(* IEC 61131-3 sources: osaicnc/ (part 2) *)

(* ---- F_SetRapidOverride.st ---- *)
(*[[
    UserText1= "V15.7",
]]*)
FUNCTION F_SetRapidOverride : DWORD
(*
F ***************************************************************************************
F * File name    : F_SetRapidOverride.st                                                *
F * Description  : Set Rapid override request from PLC, works like the system function  *
F *                block with three more possibility: the request can be applyed to all *
F *                processes, one flag permit to decide if the request is comparable    *
F *                to an operator request (like a console) and can be refused by the    *
F *                filter task, another flag enable the modification of the override    *
F *                value in the filter task (for example to align at the predefined     *
F *                steps).                                                              *
F ***************************************************************************************
F * Product line : OpenControl                                                          *
F * Enviroment   : PLC Application                                                      *
F * Component    :                                                                      *
F *                                                                                     *
F * ----------------------------------------------------------------------------------- *
F *                                                                                     *
F *   Author        date        comments                                                *
F *                                                                                     *
F *   Scapolan      23-05-16    Function creation                                       *
F *                                                                                     *
F * ----------------------------------------------------------------------------------- *
F *                                                                                     *
F * Input        :  iiExecMode          INT                                             *
F *                     Command execution modality: MODE_NOWAIT, MODE_WAIT              *
F *                                                                                     *
F *                 iiProc              INT                                             *
F *                     Process number 1..24 or -1 (ciProcAll) to request to all        *
F *                     processes.                                                      *
F *                                                                                     *
F *                 iiLastProc          INT                                             *
F *                     Last process number, used only if the request is for all        *
F *                     processes.                                                      *
F *                                                                                     *
F *                 iiNoProc            INT                                             *
F *                     Process number to skip if the request is for all processes,     *
F *                     0 to apply to every processes.                                  *
F *                                                                                     *
F *                 iiPercent           INT                                             *
F *                     New override value 10000=100%                                   *
F *                                                                                     *
F *                 iOpConsole          BOOL                                            *
F *                     Console flag, the request is comparable to an operator console, *
F *                     can be rfeused by filter task                                   *
F *                                                                                     *
F *                 iOpAdjust           BOOL                                            *
F *                     Enable modification (Adjust) of override value from PLC request *
F *                                                                                     *
F * Return       :  DWORD                                                               *
F *                     SetRapidOverride function block return code                     *
F *                                                                                     *
F * Global used  :  gPlcConOvrR          array [0..ciMaxProc] of bool                          *
F *                     Set Rapid override request from Plc console ambient memory      *
F *                                                                                     *
F *                 gPlcConAdjR          array [0..ciMaxProc] of BOOL                          *
F *                     Enable the modification of the override value in the filter     *
F *                     task (for example to align at the predefined steps)             *
F *                                                                                     *
F ***************************************************************************************

	Example for program use

\* Set Rapid override request from PLC, works like the system function block with two more possibility:
	the request can be applyed to all processes, one flag permit to decide if the request is comparable
	to an operator request (like a console) and can be refused by the filter task, another flag enable the
	modification of the override value in the filter task (for example to align at the predefined steps). */

llRetCode	:= F_SetRapidOverride(
	iiExecMode,		\* IN	INT		Command execution modality: MODE_NOWAIT, MODE_WAIT */
	iiProc,			\* IN	INT		Process number 1..24 or -1 (ciProcAll) to request to all processes */
	iiLastProc,		\* IN	INT		Last process number, used only if the request is for all processes */
	iiNoProc,		\* IN	INT		Process number to skip if the request is for all processes, 0 to apply to every processes */
	iiPercent,		\* IN	INT		New override value 10000=100% */
	iOpConsole,		\* IN	BOOL	Console flag, the request is comparable to an operator console, can be rfeused by filter task */
	iOpAdjust);		\* IN	BOOL	Enable modification (Adjust) of override value from this PLC request */

\* Example to apply the request only at the selected process with the filter enabled, the 3rd and 4th input data are not used,
	the override value are not modified in the filter task */
llRetCode	:= F_SetRapidOverride(MODE_NOWAIT, SI_PROCSEL, MI_LastProc, 0 \*iiNoProc*/, liOverride, true \*iOpConsole*/, false \*iOpAdjust*/);

\* Example to apply the request to every existing process with the filter enabled,
	but the override value are not modified in the filter task */
llRetCode	:= F_SetRapidOverride(MODE_NOWAIT, ciProcAll, MI_LastProc, 0 \*iiNoProc*/, liOverride, true \*iOpConsole*/, false \*iOpAdjust*/);

\* Example to apply the request to every existing process, except the process number 1, with the filter enabled,
	but the override value are not modified in the filter task */
llRetCode	:= F_SetRapidOverride(MODE_NOWAIT, ciProcAll, MI_LastProc, 1 \*iiNoProc*/, liOverride, true \*iOpConsole*/, false \*iOpAdjust*/);
*)

	#IMPORT  "GvU_Variable.gvl"
	#IMPORT  "Gv_Allprocess.gvl"

VAR_INPUT
	iiProc		: int;	(* Process number 1..24 or -1 (ciProcAll) to request to all processes *)
	iiPercent	: int;	(* New override value 10000=100% *)
	iOpConsole	: bool;	(* Console flag, the request is comparable to an operator console, can be rfeused by filter task *)
	iOpAdjust	: bool;	(* Enable modification (Adjust) of override value from PLC request *)
END_VAR

VAR
	llExecStatus	: dword;	(* Function block execution status, not used *)
END_VAR;

gPlcConOvrR[iiProc]	:= iOpConsole;	(* Plc console ambient memory *)
gPlcConAdjR[iiProc]	:= iOpAdjust;	(* Enable modification (Adjust) of override value from PLC request *)
F_SetRapidOverride	:= SetRapidOverride(MODE_NOWAIT, llExecStatus, iiProc, iiPercent);

END_FUNCTION

(* ---- F_SetResetProcMsg.st ---- *)
(*[[
    UserText1= "V15.7",
]]*)
(*
F ***************************************************************************************
F * File name	: F_SetResetProcMsg.st													*
F * Description	: Set/Reset second Gestop												*
F *				  When the Gestop signal ( fast output 1) is set or reset also the 		*
F *				  selected output will be set/reset										*
F ***************************************************************************************
F * Product line : OpenControl                                                          *
F * Enviroment   : PLC Application                                                      *
F * Component    :                                                                      *
F * ----------------------------------------------------------------------------------- *
F *   Author        date        comments                                                *
F *   Scapolan      19-05-16    Function creation                                       *
F * ----------------------------------------------------------------------------------- *
F * Input        :																		*
F *                 	bool															*
F ***************************************************************************************
*)
FUNCTION F_SetResetProcMsg

	#IMPORT  "Gv_AllProcess.gvl"

var_input
	ii_proc		: int;
	ii_MsgNum	: int;
	i_setreset	: bool;
end_var

var
	li_MWIndex		: int;
	li_procindex	: int;
	li_MsgIndex		: int;
	li_msg_num		: int;
	li_MsgBit		: int;
	li_mask			: word;
	li_value		: word;
end_var

(* the messagges start from 1 , the msg001 go to bit 0 of first mw *)
li_procindex := ii_proc - 1;
li_msg_num := ii_MsgNum - 1;

li_MsgIndex := li_msg_num / 16;
li_MsgBit := MOD(li_msg_num, 16);
li_mask := shl(1,li_MsgBit);
if i_setreset then
	li_value := li_mask;
else
	li_value := 0;
end_if;

if ii_proc = Current_Process then
	li_MWIndex := ciCurrProcMWMsg + li_procindex * ciNumProcMsgW + li_MsgIndex;
else
	li_MWIndex := ciFirstProcMWMsg + li_procindex * ciNumProcMsgW + li_MsgIndex;
end_if;

ArrMW[li_MWIndex] := (ArrMW[li_MWIndex] and not li_mask) or li_value;

END_FUNCTION

(* ---- F_SetSpindleOverride.st ---- *)
(*[[
    UserText1= "V15.7",
]]*)
FUNCTION F_SetSpindleOverride : DWORD
(*
F ***************************************************************************************
F * File name    : F_SetSpindleOverride.st                                              *
F * Description  : Set spindle override request from PLC, works like the system function*
F *                block with three more possibility: the request can be applyed to all *
F *                processes, one flag permit to decide if the request is comparable    *
F *                to an operator request (like a console) and can be refused by the    *
F *                filter task, another flag enable the modification of the override    *
F *                value in the filter task (for example to align at the predefined     *
F *                steps).                                                              *
F ***************************************************************************************
F * Product line : OpenControl                                                          *
F * Enviroment   : PLC Application                                                      *
F * Component    :                                                                      *
F *                                                                                     *
F * ----------------------------------------------------------------------------------- *
F *                                                                                     *
F *   Author        date        comments                                                *
F *                                                                                     *
F *   Scapolan      23-05-16    Function creation                                       *
F *                                                                                     *
F * ----------------------------------------------------------------------------------- *
F *                                                                                     *
F * Input        :  iiExecMode          INT                                             *
F *                     Command execution modality: MODE_NOWAIT, MODE_WAIT              *
F *                                                                                     *
F *                 iiProc              INT                                             *
F *                     Process number 1..24 or -1 (ciProcAll) to request to all        *
F *                     processes.                                                      *
F *                                                                                     *
F *                 iiLastProc          INT                                             *
F *                     Last process number, used only if the request is for all        *
F *                     processes.                                                      *
F *                                                                                     *
F *                 iiNoProc            INT                                             *
F *                     Process number to skip if the request is for all processes,     *
F *                     0 to apply to every processes.                                  *
F *                                                                                     *
F *                 iiPercent           INT                                             *
F *                     New override value 10000=100%                                   *
F *                                                                                     *
F *                 iOpConsole          BOOL                                            *
F *                     Console flag, the request is comparable to an operator console, *
F *                     can be rfeused by filter task                                   *
F *                                                                                     *
F *                 iOpAdjust           BOOL                                            *
F *                     Enable modification (Adjust) of override value from PLC request *
F *                                                                                     *
F * Return       :  DWORD                                                               *
F *                     SetSpindleOverride function block return code                   *
F *                                                                                     *
F * Global used  :  gPlcConOvrS          array [0..ciMaxProc] of bool                   *
F *                     Set spindle override request from Plc console ambient memory    *
F *                                                                                     *
F *                 gPlcConAdjS          array [0..ciMaxProc] of BOOL                   *
F *                     Enable the modification of the override value in the filter     *
F *                     task (for example to align at the predefined steps)             *
F *                                                                                     *
F ***************************************************************************************

	Example for program use

\* Set spindle override request from PLC, works like the system function block with two more possibility:
	the request can be applyed to all processes, one flag permit to decide if the request is comparable
	to an operator request (like a console) and can be refused by the filter task, another flag enable the
	modification of the override value in the filter task (for example to align at the predefined steps). */

llRetCode	:= F_SetSpindleOverride(
	iiExecMode,		\* IN	INT		Command execution modality: MODE_NOWAIT, MODE_WAIT */
	iiProc,			\* IN	INT		Process number 1..24 or -1 (ciProcAll) to request to all processes */
	iiLastProc,		\* IN	INT		Last process number, used only if the request is for all processes */
	iiNoProc,		\* IN	INT		Process number to skip if the request is for all processes, 0 to apply to every processes */
	iiPercent,		\* IN	INT		New override value 10000=100% */
	iOpConsole,		\* IN	BOOL	Console flag, the request is comparable to an operator console, can be rfeused by filter task */
	iOpAdjust);		\* IN	BOOL	Enable modification (Adjust) of override value from this PLC request */

\* Example to apply the request only at the selected process with the filter enabled, the 3rd and 4th input data are not used,
	the override value are not modified in the filter task */
llRetCode	:= F_SetSpindleOverride(MODE_NOWAIT, SI_PROCSEL, MI_LastProc, 0 \*iiNoProc*/, liOverride, true \*iOpConsole*/, false \*iOpAdjust*/);

\* Example to apply the request to every existing process with the filter enabled,
	but the override value are not modified in the filter task */
llRetCode	:= F_SetSpindleOverride(MODE_NOWAIT, ciProcAll, MI_LastProc, 0 \*iiNoProc*/, liOverride, true \*iOpConsole*/, false \*iOpAdjust*/);

\* Example to apply the request to every existing process, except the process number 1, with the filter enabled,
	but the override value are not modified in the filter task */
llRetCode	:= F_SetSpindleOverride(MODE_NOWAIT, ciProcAll, MI_LastProc, 1 \*iiNoProc*/, liOverride, true \*iOpConsole*/, false \*iOpAdjust*/);
*)

	#IMPORT  "GvU_Variable.gvl"
	#IMPORT  "Gv_Allprocess.gvl"

VAR_INPUT
	iiProc		: int;	(* Process number 1..24 or -1 (ciProcAll) to request to all processes *)
	iiPercent	: int;	(* New override value 10000=100% *)
	iOpConsole	: bool;	(* Console flag, the request is comparable to an operator console, can be rfeused by filter task *)
	iOpAdjust	: bool;	(* Enable modification (Adjust) of override value from PLC request *)
END_VAR

VAR
	llExecStatus	: dword;	(* Function block execution status, not used *)
END_VAR;

gPlcConOvrS[iiProc]	:= iOpConsole;	(* Plc console ambient memory *)
gPlcConAdjS[iiProc]	:= iOpAdjust;	(* Enable modification (Adjust) of override value from PLC request *)
F_SetSpindleOverride	:= SetSpindleOverride(MODE_NOWAIT, llExecStatus, iiProc, iiPercent);
if F_SetSpindleOverride<>0 then
	gPlcConOvrS[iiProc]	:= false;	(* In case of error reset the Plc console ambient memory *)
	gPlcConAdjS[iiProc]	:= false;
end_if;

END_FUNCTION

(* ---- F_Spindle_SSO.st ---- *)
(*[[
    UserText1= "V15.7",
]]*)
FUNCTION F_Spindle_SSO : lreal

	#IMPORT  "Gv_AllProcess.gvl"

var_input
	ist_spin	: St_Spindle;
END_VAR

(* Adjust programmed spindle speed with SSO *)
if ist_spin.SSO_Local > 0 then
	F_Spindle_SSO := ist_spin.MD_SpeedPro * int_to_lreal(ist_spin.SSO_Local) / 10000.0 ;
else
	F_Spindle_SSO := ist_spin.MD_SpeedPro * int_to_lreal(ArrSI[ist_spin.Spindle_process * 20 + 17]) / 10000.0 ;
end_if;

if (F_Spindle_SSO > ist_spin.Spindle_Speedmax) and not ist_spin.M_G96_SPro then
	F_Spindle_SSO := ist_spin.Spindle_Speedmax;
end_if;

END_FUNCTION

(* ---- Fb_AnalogDigital.st ---- *)
(*[[
    UserText1= "V15.7",
]]*)
FUNCTION_BLOCK Fb_AnalogDigital
VAR_INPUT
	iiMaxInp	: int;	(* Maximum input value *)
	iiMinInp	: int;	(* Minimum input value *)
	iiNumStep	: int;	(* Maximum output value *)
	idValue		:lreal;	(* Input value (analog potentiometer) *)
END_VAR

VAR_OUTPUT
	oiValue		: int;	(* Output value (new override) *)
END_VAR

VAR
	ld_valPerStep	: lreal;
	ld_valPerStep_2	: lreal;
	ld_valfiltered	: lreal;
	ld_valmemory	: lreal := -1.0;
	li_value		: int;
	li_output		: int;
	l_Init			: bool := true;
END_VAR

if l_Init then
	l_init := false;
	(* Scale calculation, only when the configuration change *)
	(* The number of step is increase by 1 because the consolle array start from 0 to NMax value *)
	ld_valPerStep := int_to_lreal(iiMaxInp - iiMinInp) / int_to_lreal(iiNumStep + 1);
	ld_valPerStep_2 := ld_valPerStep / 2.0;
end_if;

li_value := lreal_to_int(idValue);
if li_value <= iiMinInp then
	ld_valmemory := 0.0;
	li_output := 0;
elsif  li_value >= iiMaxInp then
	li_output := iiNumStep;
	ld_valmemory := int_to_lreal(iiMaxInp);
else
	ld_valfiltered := abs(idValue) - int_to_lreal(iiMinInp);
	if ld_valmemory <> ld_valfiltered then
		if  abs(ld_valmemory - ld_valfiltered) >= (ld_valPerStep_2) then
			li_output := trunc(ld_valfiltered / ld_valPerStep);
			ld_valmemory := ld_valfiltered;
		end_if;
	end_if;
end_if;

oiValue := li_output;
END_FUNCTION_BLOCK

(* ---- Fb_AnalogPotentiometer.st ---- *)
(*[[
    UserText1= "V15.7",
]]*)
FUNCTION_BLOCK Fb_AnalogPotentiometer
(*
F ***************************************************************************************
F * File name    : Fb_AnalogPotentiometer.st                                            *
F * Description  : External override potentiometer connected at analog input, with step *
F *                configuration and delay time to prevent undesired little variation.  *
F ***************************************************************************************
F * Product line : OpenControl                                                          *
F * Enviroment   : PLC Application                                                      *
F * Component    :                                                                      *
F *                                                                                     *
F * ----------------------------------------------------------------------------------- *
F *                                                                                     *
F *   Author       date      comments                                                   *
F *                                                                                     *
F *   Mazzocco     27-04-10  Function block creation                                    *
F *                                                                                     *
F * ----------------------------------------------------------------------------------- *
F *                                                                                     *
F * Input        :  iiMaxInp            INT                                             *
F *                     Maximum input value                                             *
F *                                                                                     *
F *                 iiMinInp            INT                                             *
F *                     Minimum input value                                             *
F *                                                                                     *
F *                 iiMaxOut            INT                                             *
F *                     Maximum output value                                            *
F *                                                                                     *
F *                 iiMinOut            INT                                             *
F *                     Minimum output value                                            *
F *                                                                                     *
F *                 iiStepOut           INT                                             *
F *                     Minimum variation for output value (in output signal scale)     *
F *                                                                                     *
F *                 iiStepAct           INT                                             *
F *                     Minimum variation in output signal scale that activate the      *
F *                     potentiometer                                                   *
F *                                                                                     *
F *                 iiDelay             TIME                                            *
F *                     Dealy to leave active the potentiometer when the variation are  *
F *                     little of minimum iiStepAct                                     *
F *                                                                                     *
F *                 iiValue             INT                                             *
F *                     Input value (analog potentiometer)                              *
F *                                                                                     *
F * Output       :  oiValue             INT                                             *
F *                     Output value (new override)                                     *
F *                                                                                     *
F *                 oError              BOOL                                            *
F *                     Scale value wrong (minimum value bigger then maximum or         *
F *                     division by zero)                                               *
F *                                                                                     *
F * Global used  :      Not used                                                        *
F *                                                                                     *
F ***************************************************************************************
*)

(* Example for program use
VAR
	Fb_1AnPot	:Fb_AnalogPotentiometer;	\* External override potentiometer connected at analog input */
END_VAR

\* External override potentiometer connected to analog input */
Fb_1AnPot(
	iiMaxInp	:= 2048,		\* IN	INT		Maximum input value */
	iiMinInp	:= 0,			\* IN	INT		Minimum input value */
	iiMaxOut	:= 10000,		\* IN	INT		Maximum output value */
	iiMinOut	:= 0,			\* IN	INT		Minimum output value */
	iiStepOut	:= 100,			\* IN	INT		Minimum variation for output value (in output signal scale) */
	iiStepAct	:= 200,			\* IN	INT		Minimum variation in output signal scale that activate the potentiometer */
	iiDelay		:= t#3000ms,	\* IN	TIME	Dealy to leave active the potentiometer when the variation are little of minimum iiStepAct */
	iiValue		:= liAnPot?,	\* IN	INT		Input value (analog potentiometer) */
	oiValue		=> liNewOvr?,	\* OUT	INT		Output value (new override) */
	oError		=> lErrMsg?);	\* OUT	BOOL	Scale value wrong (minimum value bigger then maximum or division by zero) *)

VAR_INPUT
	iiMaxInp	: int;	(* Maximum input value *)
	iiMinInp	: int;	(* Minimum input value *)
	iiMaxOut	: int;	(* Maximum output value *)
	iiMinOut	: int;	(* Minimum output value *)
	iiStepOut	: int;	(* Minimum variation for output value (in output signal scale) *)
	iiStepAct	: int;	(* Minimum variation in output signal scale that activate the potentiometer *)
	iiDelay		:TIME;	(* Dealy to leave active the potentiometer when the variation are little of minimum iiStepAct *)
	iiValue		: int;	(* Input value (analog potentiometer) *)
END_VAR

VAR_OUTPUT
	oiValue		: int;	(* Output value (new override) *)
	oError		: bool;	(* Scale value wrong (min value bigger then max or division by zero) *)
END_VAR

VAR
	liMaxInp	: int;	(* Maximum input value *)
	liMinInp	: int;	(* Minimum input value *)
	liMaxOut	: int;	(* Maximum output value *)
	liMinOut	: int;	(* Minimum output value *)
	liStepOut	: int;	(* Minimum variation for output value (in output signal scale) *)
	liOutNum	: int;	(* Number of output value *)
	liStepInp	: int;	(* Input step corrispondent to the configured output step *)
	liValue		: int;	(* Output value continuous calculation *)
	liDiff		: int;	(* Difference between new calculated value and active output value *)
	TON_Disable	:TON;	(* Potentiometer disable delay *)
END_VAR

(* Scale calculation, only when the configuration change *)
if iiMaxInp<>liMaxInp or iiMinInp<>liMinInp or iiMaxOut<>liMaxOut or iiMinOut<>liMinOut or
iiStepOut<>liStepOut or liOutNum=0 or oError then

	liMaxInp	:= iiMaxInp;
	liMinInp	:= iiMinInp;
	liMaxOut	:= iiMaxOut;
	liMinOut	:= iiMinOut;
	liStepOut	:= iiStepOut;

	(* Compare minimum value with maximum value and division by zero *)
	if liMaxInp<liMinInp or liMaxOut<liMinOut or liStepOut=0 then
		oError	:= true;
	else

		(* Number of output value calculation *)
		liOutNum	:= (liMaxOut - liMinOut) / liStepOut;

		if liOutNum=0 then
			oError	:= true;
		else
			(* Input step calculation *)
			liStepInp	:= (liMaxInp - liMinInp) / liOutNum;

			if liStepInp=0 then
				oError	:= true;
			else
				oError	:= false;
			end_if;

		end_if;

	end_if;

end_if;

if not oError then

	(* Output value continuous calculation *)
	liValue	:= LIMIT(liMinOut, ((iiValue - liMinInp) / liStepInp * liStepOut) + liMinOut, liMaxOut);

	(* Output difference calculation *)
	liDiff	:= oiValue - liValue;

end_if;

(* Potentiometer disable delay *)
TON_Disable(IN := ABS(liDiff)<ABS(iiStepAct), PT := iiDelay);

(* New output value activation *)
if not TON_Disable.Q and not oError then
	oiValue	:= liValue;
end_if;

END_FUNCTION_BLOCK

(* ---- Fb_AuxAxis.st ---- *)
(*[[
    UserText1= "V15.7",
]]*)
FUNCTION_BLOCK Fb_AuxAxis
	#IMPORT  "Gv_AllProcess.gvl"
(*
F ***************************************************************************************
F * File name    : Fb_AuxAxis.st                                                        *
F * Description  : PLC single axis handling, tipically a rollover rotary tool magazine  *
F ***************************************************************************************
F * Product line : OpenControl                                                          *
F * Enviroment   : PLC Application                                                      *
F * Component    :                                                                      *
F *                                                                                     *
F * ----------------------------------------------------------------------------------- *
F *                                                                                     *
F *   Author       date      comments                                                   *
F *                                                                                     *
F *   Mazzocco     17-03-10  Creation Fb_AuxAxis                                        *
F *   Mazzocco     06-10-10  Add sequential cycle phase number in output for diagnostic *
F *   Mazzocco     22-06-11  Add feed-hold management.                                  *
F *   Mazzocco     09-09-11  Add moving property specification, change requested        *
F *                          position variable type from input to input/output,         *
F *                          modified override scale to adapt at new release 2.1        *
F *                          (100%=10000 and not 100), remove included interpolator     *
F *                          management                                                 *
F *   Paglia L.	   13-10-11  Added Input "iiValFeed" for "Work" type movement           *
F *   Mazzocco     26-04-12  Optimized property and override management.                *
F *   Scapolan     08-03-18  Optimized use of gst_axisinfo                              *
F *                                                                                     *
F * ----------------------------------------------------------------------------------- *
F *                                                                                     *
F * Input        :  iFbEnable           BOOL                                            *
F *                     Function block enable                                           *
F *                                                                                     *
F *                 iReset              BOOL                                            *
F *                     Reset error request                                             *
F *                                                                                     *
F *                 ibProperty          BYTE                                            *
F *                     Axis movement property definition: bit 0 MODE_INCR incremental, *
F *                     bit 1 MODE_ROLLOPT rollover optimized, bit 2 MODE_NOFEED don't  *
F *                     considerate in feed calculation                                 *
F *                                                                                     *
F *                 iiTypeFeed          INT                                             *
F *                     Feed type: 0 MODE_RAPID, 1 MODE_WORK, 2 MODE_FEED_t,            *
F *                     3 MODE_FEED_1T                                                  *
F *                                                                                     *
F *                 idValue             LREAL                                           *
F *                     Feed Value: units pe minut. Only for working movement           *
F *                                                                                     *
F *                 iiOverPerc          INT                                             *
F *                     Feed override percent                                           *
F *                                                                                     *
F *                 iiAxisID            INT                                             *
F *                     Auxiliary axis identifier                                       *
F *                                                                                     *
F *                 iiProc              INT                                             *
F *                     Process number                                                  *
F *                                                                                     *
F *                 iSt_InterpInfo      InterpInfo_Struct                               *
F *                     PLC inerpolator info structure                                  *
F *                                                                                     *
F *                 iiInterpID          INT                                             *
F *                     Interpolator number                                             *
F *                                                                                     *
F *                 iForceHome          BOOL                                            *
F *                     Homing cycle forced at every movement                           *
F *                                                                                     *
F * Input/Output :  ioReqMove           BOOL                                            *
F *                     Movement request                                                *
F *                                                                                     *
F *                 iodPosition         LREAL                                           *
F *                     Requested position                                              *
F *                                                                                     *
F *                 ioiAck              INT                                             *
F *                     Event task need acknowledge:                                    *
F *                         1 M function at movement end,                               *
F *                         2 M function starting movement,                             *
F *                         3 Pseudo axes at movement end.                              *
F *                         4 Pseudo axes starting movement,                            *
F *                                                                                     *
F * Output       :  oEndSignal          BOOL                                            *
F *                     Movement completed                                              *
F *                                                                                     *
F *                 oMoving             BOOL                                            *
F *                     Auxiliary axis is moving                                        *
F *                                                                                     *
F *                 oHoming             BOOL                                            *
F *                     Auxiliary axis is homing                                        *
F *                                                                                     *
F *                 oSt_AxisInfo        AxisInfo_Struct                                 *
F *                     Axis info structure                                             *
F *                                                                                     *
F *                 oiPhase             INT                                             *
F *                     Movement sequential cycle phase number                          *
F *                                                                                     *
F *                 olRetCode           DWORD                                           *
F *                     Function block return code                                      *
F *                                                                                     *
F * Global used  :      Not used                                                        *
F *                                                                                     *
F * Attention    :  Use this FB directly in the logic program, don't inside a cycle     *
F *                 (IF, FOR, etc.), is the same for all the macro function block with  *
F *                 the iFbEnable input.                                                *
F *                                                                                     *
F ***************************************************************************************
*)

(* Example for program use
VAR
	Fb_1AuxAxis	:Fb_AuxAxis;	\* PLC single axis handling */
END_VAR

\* PLC single axis handling */
Fb_1AuxAxis(
	iFbEnable		:= M_EnabDone,		\* IN	BOOL	Function block enable */
	iReset			:= M_Reset?,		\* IN	BOOL	Reset error request */
	ibProperty		:= MODE_?,			\* IN	BYTE	Axis movement property definition: bit 0 MODE_INCR incremental, bit 1 MODE_ROLLOPT rollover optimized, bit 2 MODE_NOFEED don't considerate in feed calculation */
	iiTypeFeed		:= MODE_?,			\* IN	INT		Feed type: 0 MODE_RAPID, 1 MODE_WORK, 2 MODE_FEED_t, 3 MODE_FEED_1T */
	idValue			:= 0.0,				\* IN	LREAL	Feed value for working movement */
	iiOverPerc		:= SI_?Rap,			\* IN	INT		Feed override percent */
	iiAxisID		:= GI_Id_?,			\* IN	INT		Auxiliary axis identifier */
	iiProc			:= ciProc_?,		\* IN	INT		Process number */
	iSt_InterpInfo  := gSt_InterpInfo[MI_InterpId_?],	\* IN  InterpInfo_Struct	PLC inerpolator info structure */
	iiInterpID		:= MI_InterpId_?,	\* IN	INT		Interpolator number */
	iForceHome		:= gSt_PlcCfg.Ah_Aux_Home,			\* IN	BOOL	Homing cycle forced at every movement */

	ioReqMove		:= M_Req_Mov_?,		\* I/O	BOOL	Movement request */
	iodPosition		:= MD_ReqPos_?,		\* I/O	LREAL	Requested position */
	ioiAck			:= MI_Ack_Mov_?,	\* I/O	INT		Event task need acknowledge: 1 M function at movement end, 2 M function starting movement, 3 Pseudo axes at movement end, 4 Pseudo axes starting movement */

	oEndSignal		=> ,					\* OUT	BOOL	Movement completed */
	oMoving			=> M_AxesMovC[GI_Id_?],	\* OUT	BOOL	Auxiliary axis is moving */
	oHoming			=> M_Home_?,			\* OUT	BOOL	Auxiliary axis is homing */
	oSt_AxisInfo	=> gSt_AxisInfo[GI_Id_?],			\* OUT	AxisInfo_Struct		Axis info structure */
	oiPhase			=> ,					\* OUT	INT		Movement sequential cycle phase number */
	olRetCode		=> llRetCode?);			\* OUT	DWORD	Function block return code *)

VAR_INPUT
	iFbEnable		: bool;		(* Function block enable *)
	iReset			: bool;		(* Function block reset error request *)
	ibProperty		: byte;		(* Axis movement property definition: bit 0 MODE_INCR incremental, bit 1 MODE_ROLLOPT rollover optimized, bit 2 MODE_NOFEED don't considerate in feed calculation *)
	iiTypeFeed		: int;		(* Feed type: 0 MODE_RAPID, 1 MODE_WORK, 2 MODE_FEED_t, 3 MODE_FEED_1T *)
	idValue			: lreal;	(* Feed value *)
	iiOverPerc		: int;		(* Feed override percent *)
	iiAxisID		: int;		(* Auxiliary axis identifier *)
	iiProc			: int;		(* Process number *)
	iSt_InterpInfo  : InterpInfo_Struct;		(* PLC inerpolator info structure *)
	iiInterpID		: int;		(* Interpolator number *)
	iForceHome		: bool;		(* Homing cycle forced at every movement *)
END_VAR

VAR_IN_OUT
	ioReqMove		: bool;		(* Movement request *)
	iodPosition		: lreal;	(* Requested position *)
	ioiAck			: int;		(* Event task need acknowledge: 1 M function at movement end, 2 M function starting movement, 3 Pseudo axes at movement end, 4 Pseudo axes starting movement *)
END_VAR

VAR_OUTPUT
	oEndSignal		: bool;		(* Movement completed *)
	oMoving			: bool;		(* Auxiliary axis is moving *)
	oHoming			: bool;		(* Auxiliary axis is homing *)
	oSt_AxisInfo	: AxisInfo_Struct;		(* axis info structure *)
	oiPhase			: int;		(* Movement sequential cycle phase number *)
	olRetCode		: dword;	(* Return code of the function block *)
END_VAR

VAR
	llRetCodeSAP	: dword;	(* Set axis property function block return code *)
	llRetCodeSFO	: dword;	(* Set feed override function block return code *)
	llRetCodeGM 	: dword;	(* Move function block return code *)
	llRetCodeACK	: dword;	(* Acknowledge strobe function block return code *)
	llExecStatus	: dword;	(* Function block execution status not used *)
	lbMemProp		: BYTE;		(* Axis movement property memory *)
	lbActProp		: BYTE;		(* Axis movement active property *)
	lErrSAP			: BOOL	:= true;	(* Error in setting axis poperty , to generate a refresh request *)
	lErrSFO			: BOOL	:= true;	(* Error in setting axis override, to generate a refresh request *)
	liMemOver		: int;		(* Feed override memory *)
	lAckM			: bool;		(* M function event task need acknowledge at the end of the movement *)
	lAckP			: bool;		(* Pseudo axes event task need acknowledge at the end of the movement *)
	ldPosition		: lreal;	(* Requested position memory *)
	lEndHome		: bool;		(* Homing movement completed *)
	liInterpId		: int;		(* Interpolator number memory *)
	liAxisId		: int;		(* Axis identifier number memory *)

	lSt_Feed		:FeedDescr_Struct;
	(*	TypeFeed	: int;	- Feed type					-
		Value		:lreal;	- Feed value				-
		Accel		:lreal;	- Target acceleration != 0	-
		Decel		:lreal;	- Target deceleration != 0	-
		Jerk		:lreal;	- Target jerk != 0			-
		VelOnlyLin	: bool;	- Vel for linear axes only	-	*)
END_VAR

(* Interpolator reset completed, delete movement flag *)
if iSt_InterpInfo.TaskSts = INT_ST_IDLE or iSt_InterpInfo.TaskSts = INT_ST_ERR or
iSt_InterpInfo.TaskSts = INT_ST_EMG then
	oMoving	:= false;	(* Auxiliary axis is moving *)
	oHoming	:= false;	(* Auxiliary axis is homing *)
end_if;

if iFbEnable then

	(* Refresh axis info *)
	oSt_AxisInfo := Gst_AxisInfo[iiAxisId];

	if iiInterpID>0 and iiInterpID<41 and iiAxisId>0 and iiAxisId<65 and olRetCode=0 then

		(* Check axes and interpolator number value *)
		if liInterpId<>iiInterpID or liAxisId<>iiAxisId then
			liInterpID	:= iiInterpID;
			liAxisId	:= iiAxisId;
			lErrSap	:= true;
			lErrSfo	:= true;
		end_if;

		if oiPhase<>0 then
			(* Set axis property *)
			if llRetCodeSAP=0 and (ibProperty<>lbMemProp or lErrSAP) then
				if iSt_InterpInfo.TaskSts = INT_ST_IDLE and not iReset then
					lbMemProp := ibProperty;

					if (oSt_AxisInfo.AxType and _AX_ROLLOVER)<>0 then
						lbActProp := lbMemProp;
						llRetCodeSAP := GMC_SetAxisProperty(MODE_NOWAIT, llExecStatus, iiInterpID, lbActProp, iiAxisId);
					else
						(* Delete the rollover optimized bit for not rollover axis *)
						lbActProp	:= lbMemProp and 16#00FD;
						llRetCodeSAP	:= GMC_SetAxisProperty(MODE_NOWAIT, llExecStatus, iiInterpID,
							lbActProp, iiAxisId);
					end_if;

					lErrSAP	:= llRetCodeSAP<>0;	(* Refresh request in case of error *)
				end_if;
			end_if;

			(* Set override *)
			if llRetCodeSFO=0 and (iiOverPerc<>liMemOver or lErrSFO) then
				liMemOver		:= iiOverPerc;
				llRetCodeSFO	:= GMC_SetFeedOverride(MODE_NOWAIT, llExecStatus, iiInterpID,
					iiAxisId, liMemOver);

				lErrSFO	:= llRetCodeSFO<>0;	(* Refresh request in case of error *)
			end_if;
		end_if;

		(* Movement phase *)
		if llRetCodeGM=0 and iSt_InterpInfo.TaskSts = INT_ST_IDLE and (oiPhase=0 or (lbMemProp=ibProperty and
			oSt_AxisInfo.ProgrMode=lbActProp and iiOverPerc=liMemOver and oSt_AxisInfo.Override=INT_TO_WORD(iiOverPerc) and
			not lErrSap and not lErrSfo)) and
			(oSt_AxisInfo.AxisHwSts and _ZEROASS)=0 and liInterpId=iiInterpID and liAxisId=iiAxisId then

			case oiPhase of

				00:	(* Wait movement request *)
					if ioReqMove then
						oEndSignal	:= false;	(* Reset end movement flag *)
						ioReqMove	:= false;	(* Reset movement request *)
						ldPosition	:= iodPosition;	(* Store requested position *)
						liMemOver	:= -1;	(* Update override *)

						(* Reset acknowledge request memory *)
						lAckM	:= false;
						lAckP	:= false;

						case ioiAck of
							01:	(* M function event task need acknowledge at the end of the movement *)
								lAckM	:= true;

							02:	(* M function event task need acknowledge at the beginning of the movement *)
								ioiAck			:= 0;
						        llRetCodeACK	:= AckStrobePProgram(iiProc, f_M_FUNCTION, Ack);

							03:	(* Pseudo axes event task need acknowledge at the end of the movement *)
								lAckP	:= true;

							04:	(* Pseudo axes event task need acknowledge at the beginning of the movement *)
								ioiAck			:= 0;
						        llRetCodeACK	:= AckStrobePProgram(iiProc, f_PSEUDO_AX_FUNCTION, Ack);
						end_case;

						ioiAck	:= 0;	(* Reset acknowledge request in any case *)

						(* Check axis referred *)
						if (oSt_AxisInfo.AxisHwSts and _HC_DONE)=0 or iForceHome then
							oHoming	:= true;
							oiPhase	:= 1;
						else
							lSt_Feed.TypeFeed	:= iiTypeFeed;
							lSt_Feed.Value	:= idValue;

							llRetCodeGM	:= GMC_Move(MODE_NOWAIT, llExecStatus, iiInterpID, oEndSignal,
								lSt_Feed, iiAxisId, ldPosition);

							oMoving	:= true;	(* Auxiliary axis is moving *)
							oiPhase	:= 4;	(* Auxiliary axis is homing *)
						end_if;
					end_if;

				01: (* Homing request *)
					lEndHome	:= false;
					llRetCodeGM	:= GMC_Homing(MODE_NOWAIT, llExecStatus, iiInterpID, lEndHome, iiAxisId);
					oMoving	:= true;	(* Auxiliary axis is moving *)
					oiPhase	:= oiPhase + 1;

				02:	(* Wait homing movement completed *)
					if lEndHome then
						oMoving	:= false;	(* Auxiliary axis is moving *)
						oHoming	:= false;	(* Auxiliary axis is homing *)
						oiPhase	:= oiPhase + 1;
					end_if;

				03:	(* Movement request *)
					if (oSt_AxisInfo.AxisHwSts and _HC_DONE) <> 0 then
						lSt_Feed.TypeFeed := iiTypeFeed;
						lSt_Feed.Value := idValue;

						llRetCodeGM	:= GMC_Move(MODE_NOWAIT, llExecStatus, iiInterpID, oEndSignal, lSt_Feed, iiAxisId, ldPosition);

						oMoving	:= true;	(* Auxiliary axis is moving *)
						oiPhase	:= oiPhase + 1;
					end_if;

				04:	(* Wait movement completed *)
					if oEndSignal then
						if lAckM then	(* Release M function event task *)
							lAckM			:= false;
					        llRetCodeACK	:= AckStrobePProgram(iiProc, f_M_FUNCTION, Ack);
						end_if;

						if lAckP then	(* Release pseudo axes event task *)
							lAckP			:= false;
					        llRetCodeACK	:= AckStrobePProgram(iiProc, f_PSEUDO_AX_FUNCTION, Ack);
						end_if;

						oMoving	:= false;	(* Auxiliary axis is moving *)
						oiPhase	:= 0;
					end_if;

			end_case;

		end_if;

	end_if;

	(* return code management *)
	if olRetCode=0 then
		if llRetCodeSAP<>0 then
			olRetCode	:= llRetCodeSAP;
		elsif llRetCodeSFO<>0 then
			olRetCode	:= llRetCodeSFO;
		elsif llRetCodeGM<>0 then
			olRetCode	:= llRetCodeGM;
		elsif llRetCodeACK<>0 then
			olRetCode	:= llRetCodeACK;
		end_if;
	end_if;

end_if;

(* reset management *)
if iReset then
	llRetCodeSAP	:= 0;
	llRetCodeSFO	:= 0;
	llRetCodeGM		:= 0;
	llRetCodeACK	:= 0;
	olRetCode		:= 0;
	oEndSignal		:= false;	(* Reset end movement flag *)
	ioReqMove		:= false;	(* Reset movement request *)
	ioiAck			:= 0;
	oiPhase			:= 0;
	lbMemProp		:= 0;
end_if;

END_FUNCTION_BLOCK

(* ---- Fb_AuxSpindle.st ---- *)
(*[[
    UserText1= "V15.7",
]]*)
FUNCTION_BLOCK Fb_AuxSpindle

	#IMPORT  "Gv_AllProcess.gvl"
	#IMPORT  "Gv_Functionblock.gvl"

(*
F ***************************************************************************************
F * File name    : Fb_AuxSpindle.st                                                     *
F * Description  : PLC single digital spindle handling 									*
F ***************************************************************************************
F * Product line : OpenControl                                                          *
F * Enviroment   : PLC Application                                                      *
F * Component    :                                                                      *
F * ----------------------------------------------------------------------------------- *
F *                                                                                     *
F *   Author       date      comments                                                   *
F *                                                                                     *
F *   Scapolan     24-10-16  Creation                                                   *
F *                                                                                     *
F * ----------------------------------------------------------------------------------- *
F *                                                                                     *
F * Input        :  iFbEnable           BOOL                                            *
F *                     Function block enable                                           *
F *                                                                                     *
F *                 iReset              BOOL                                            *
F *                     Reset error request                                             *
F *                                                                                     *
F *                                                                                     *
F *                 iiOverPerc          INT                                             *
F *                     Feed override percent                                           *
F *                                                                                     *
F *                 iiAxisID            INT                                             *
F *                     Auxiliary axis identifier                                       *
F *                                                                                     *
F *                 iiProc              INT                                             *
F *                     Process number                                                  *
F *                                                                                     *
F *                 iw_Tasksts			word				                            *
F *                     PLC inerpolator status			                                *
F *                                                                                     *
F *                 iiInterpID          INT                                             *
F *                     Interpolator number                                             *
F *                                                                                     *
F *                                                                                     *
F * Input/Output :  ioReqMove           BOOL                                            *
F *                     Movement request                                                *
F *                                                                                     *
F *                 iodPosition         LREAL                                           *
F *                     Requested position                                              *
F *                                                                                     *
F *                 ioiAck              INT                                             *
F *                     Event task need acknowledge:                                    *
F *                         1 M function at movement end,                               *
F *                         2 M function starting movement,                             *
F *                         3 Pseudo axes at movement end.                              *
F *                         4 Pseudo axes starting movement,                            *
F *                                                                                     *
F * Output       :  oEndSignal          BOOL                                            *
F *                     Movement completed                                              *
F *                                                                                     *
F *                 oMoving             BOOL                                            *
F *                     Auxiliary axis is moving                                        *
F *                                                                                     *
F *                 oHoming             BOOL                                            *
F *                     Auxiliary axis is homing                                        *
F *                                                                                     *
F *                 gSt_AxisInfo[iiAxisID].        AxisInfo_Struct                                 *
F *                     Axis info structure                                             *
F *                                                                                     *
F *                 oiPhase             INT                                             *
F *                     Movement sequential cycle phase number                          *
F *                                                                                     *
F *                 olRetCode           DWORD                                           *
F *                     Function block return code                                      *
F *                                                                                     *
F * Global used  :      Not used                                                        *
F *                                                                                     *
F * Attention    :  Use this FB directly in the logic program, don't inside a cycle     *
F *                 (IF, FOR, etc.), is the same for all the macro function block with  *
F *                 the iFbEnable input.                                                *
F *                                                                                     *
F ***************************************************************************************
*)

(* Example for program use
VAR
	Fb_1AuxAxis	:Fb_AuxAxis;	\* PLC single axis handling */
END_VAR

\* PLC single axis handling */
Fb_1AuxAxis(
	iFbEnable		:= M_EnabDone,		\* IN	BOOL	Function block enable */
	iReset			:= M_Reset?,		\* IN	BOOL	Reset error request */
	iiOverPerc		:= SI_?Rap,			\* IN	INT		Feed override percent */
	iiAxisID		:= GI_Id_?,			\* IN	INT		Auxiliary axis identifier */
	iw_Tasksts		:= gSt_InterpInfo[MI_InterpId_?].TaskSts,	\* IN  InterpInfo_Struct	PLC inerpolator info structure */
	iiInterpID		:= MI_InterpId_?,	\* IN	INT		Interpolator number */

	oEndSignal		=> ,					\* OUT	BOOL	Movement completed */
	oMoving			=> M_AxesMovC[GI_Id_?],	\* OUT	BOOL	Auxiliary axis is moving */
	oHoming			=> M_Home_?,			\* OUT	BOOL	Auxiliary axis is homing */
	oiPhase			=> ,					\* OUT	INT		Movement sequential cycle phase number */
	olRetCode		=> llRetCode?);			\* OUT	DWORD	Function block return code *)

VAR_INPUT
	iFbEnable		: bool;	(* Function block enable *)
	iReset			: bool;	(* Function block reset error request *)
	iiOverPerc		: int;	(* Feed override percent *)
	iiAxisID		: int;	(* Auxiliary axis identifier *)
	ii_proc			: int;	(* Auxiliary axis identifier *)
	iw_TaskSts		: word; (* PLC inerpolator status *)
	iiInterpID		: int;	(* Interpolator number *)
END_VAR

VAR_OUTPUT
	oMoving			: bool;	(* Auxiliary axis is moving *)
	olRetCode		: dword;	(* Return code of the function block *)
END_VAR

VAR
	ll_RetCode		: dword;
	llExecStatus	: dword;	(* Function block execution status not used *)
	liMemOver		: array [0..MAX_ASSI] of int;	(* Feed override memory *)

	li_Phase		: int;
	li_Phases		: array [0..MAX_ASSI] of int;
	l_enabrun		: array [0..MAX_ASSI] of bool;
	l_EndSignal		: array [0..MAX_ASSI] of bool;
	l_init			: bool := 1;
END_VAR

if iFbEnable or iReset then

	oMoving	:= true;

	(* Set override *)
	if (iiOverPerc <> liMemOver[iiAxisID]) or l_init then
		l_init := false;
		liMemOver[iiAxisID] := iiOverPerc;
		ll_RetCode := GMC_SetFeedOverride(MODE_NOWAIT, llExecStatus, iiInterpID, iiAxisID, liMemOver[iiAxisID]);
	end_if;

	li_Phase := li_Phases[iiAxisID];
	case li_Phase of

		0:
			(* Only if the axis spindle is released from process we can move it *)
			if iReset then
				if l_enabrun[iiAxisID] then
					Fb_Enab_One_Axis(iFbEnable := False, ii_AxId := iiAxisID,ii_proc := ii_proc);
					l_enabrun[iiAxisID] := false;
				end_if;
				li_Phase := li_Phase + 1;
				oMoving	:= false;

			elsif gSt_AxisInfo[iiAxisID].SharingProc <> 0 and iFbEnable then

				if not M_AxisEnabDisab[iiAxisID] or l_enabrun[iiAxisID] then
					Fb_Enab_One_Axis(iFbEnable := true, ii_AxId := iiAxisID, ii_proc := ii_proc );
					l_enabrun[iiAxisID] := true;
					if Fb_Enab_One_Axis.oDone then
						Fb_Enab_One_Axis(iFbEnable := False, ii_AxId := iiAxisID, ii_proc := ii_proc );
						l_enabrun[iiAxisID] := false;
					end_if;
				end_if;
				if not l_enabrun[iiAxisID] and iw_TaskSts = INT_ST_IDLE then
					ll_RetCode	:=  GMC_MoveJog(MODE_NOWAIT, llExecStatus, iiInterpID, l_EndSignal[iiAxisID], MAN_HWLIMSTOP, iiAxisID);
					li_Phase := li_Phase + 1;
				end_if;

			else
				oMoving	:= false;
			end_if;

		1:
			if iReset then
				if iw_TaskSts = INT_ST_IDLE or iw_TaskSts = INT_ST_ERR or iw_TaskSts = INT_ST_EMG or iw_TaskSts = INT_ST_HOLD then
					if M_AxisEnabDisab[iiAxisID] or l_enabrun[iiAxisID] then
						Fb_Disable_One_Axis(iFbEnable := true, ii_AxId := iiAxisID, ii_proc := ii_proc);
						l_enabrun[iiAxisID] := true;
						if Fb_Disable_One_Axis.oDone then
							Fb_Disable_One_Axis(iFbEnable := false, ii_AxId := iiAxisID, ii_proc := ii_proc);
							l_enabrun[iiAxisID] := false;
							li_Phase := 0;
							oMoving := false;
						end_if;
					end_if;
				end_if;
			else
				li_Phase := 0;
				oMoving := false;
			end_if;
	end_case;

	li_Phases[iiAxisID] := li_Phase;
end_if;

(* reset management *)

END_FUNCTION_BLOCK

(* ---- Fb_Button.st ---- *)
(*[[
    UserText1= "V15.7",
]]*)
FUNCTION_BLOCK Fb_Button

(*
F ***************************************************************************************
F * File name    : FB_Button.st                                                         *
F * Description  : Button or selector interface with delay and manteined or On/Off      *
F *                functionality                                                        *
F ***************************************************************************************
F * Product line : OpenControl                                                          *
F * Enviroment   : PLC Application                                                      *
F * Component    :                                                                      *
F *                                                                                     *
F * ----------------------------------------------------------------------------------- *
F *                                                                                     *
F *   Author        date        comments                                                *
F *                                                                                     *
F *   Scapolan      08-02-17    Creation Function Block                                 *
F * ----------------------------------------------------------------------------------- *
F *                                                                                     *
F * Input        :  iFbEnable	BOOL	Function block enable							*
F *                 iButOn		BOOL	Physical button (ON request)					*
F *                 iActOn		BOOL													*
F *                     Flag to check actual condition (ON), used only with iMode=TRUE  *
F *                     to choose the OFF or ON request                                 *
F *                                                                                     *
F *                 iMode		BOOL	Working mode									*
F *                     FALSE Manteined, ON request pressing button, OFF request        *
F *                           releasing button                                          *
F *                     TRUE  ON/OFF, press button and request change from ON to OFF or *
F *                           from OFF to ON, release button and nothing appen          *
F *                                                                                     *
F * Input/Output :  ioOn                 BOOL                                           *
F *                     ON request, can be resetted from the PLC                        *
F *                                                                                     *
F *                 ioOff                BOOL                                           *
F *                     OFF request, can be resetted from the PLC                       *
F *                                                                                     *
F * Global used  :      not used                                                        *
F *                                                                                     *
F * Attention    :  Use this FB directly in the logic program, don't inside a cycle     *
F *                 (IF, FOR, etc.), is the same for all the macro function block with  *
F *                 the iFbEnable input.                                                *
F *                                                                                     *
F ***************************************************************************************

    Example for program use

VAR
	FB_1Button	:FB_Button;	\* Button or selector interface with delay and manteined or On/Off functionality */
END_VAR

\* Button or selector interface with delay and manteined or On/Off functionality */
FB_1Button(
	iFbEnable	:= ,			\* IN	BOOL	Function block enable */
	iButOn		:= I_But_?,		\* IN	BOOL	Physical button (ON request) */
	iActOn		:= lMemButOn,	\* IN	BOOL	Flag to check actual condition (ON), used only with iMode=TRUE to choose the OFF or ON request */
	iMode		:= ,			\* IN	BOOL	Working mode:
									FALSE Manteined, ON request pressing button, OFF request releasing button
									TRUE  ON/OFF, press button and request change from ON to OFF or from OFF to ON, release button and nothing appen */
	ioOn		:= lButOn,		\* I/O	BOOL	ON request, can be resetted from the PLC */
	ioOff		:= lButOff);	\* I/O	BOOL	OFF request, can be resetted from the PLC *)

VAR_INPUT
	iFbEnable	: bool;	(* Function block enable *)
	iButOn		: bool;	(* Physical button *)
	iActOn		: bool;	(* Flag to check actual condition (ON), used only with iMode=TRUE to choose the OFF or ON request *)
	iMode		: bool;	(* Working mode:	FALSE Manteined, ON request pressing button, OFF request releasing button
											TRUE  ON/OFF, press button and request change from ON to OFF or from OFF to ON, release button and nothing appen *)
END_VAR

VAR_IN_OUT
	ioOn	: bool;	(* ON request, can be resetted from the PLC *)
	ioOff	: bool;	(* OFF request, can be resetted from the PLC *)
END_VAR

VAR
	RT_But		:R_TRIG;	(* Press button trigger *)
	lReqOn		: bool;		(* On request memory *)
	lReqOff		: bool;		(* Off request memory *)
	RT_On		:R_TRIG;	(* On request output *)
	RT_Off		:R_TRIG;	(* Off request output *)
END_VAR

(* Press button trigger *)
RT_But(CLK := iButOn);

if iFbEnable then

	if iMode then
		(* ON/OFF mode, press button and request change from ON to OFF or from OFF to ON,
			release button and nothing appen *)

		(* Pressing button check actual condition and store the ON/OFF request *)
		if RT_But.Q then
			if iActOn then
				(* Off request *)
				lReqOn	:= false;
				lReqOff	:= true;
			else
				(* On request *)
				lReqOn	:= true;
				lReqOff	:= false;
			end_if;
		end_if;

		(* Releasing button delete request *)
		if not iButOn then
			lReqOn	:= false;
			lReqOff	:= false;
		end_if;
	else
		(* Manteined mode, ON request pressing button, OFF request releasing button *)
		lReqOn	:= iButOn;		(* if button press lRepOn=true, lReqOff=false *)
		lReqOff	:= not iButOn;	(* if button release lRepOn=false, lReqOff=true *)
	end_if;

else
	lReqOn	:= false;
	lReqOff	:= false;
	ioOn	:= false;
	ioOff	:= false;
end_if;

(* On request after delay *)
RT_On(CLK := not lReqOff and lReqOn);
if RT_On.Q then
	ioOn	:= true;
	ioOff	:= false;
end_if;

(* Off request after delay *)
RT_Off(CLK := lReqOff and not lReqOn);
if RT_Off.Q then
	ioOn	:= false;
	ioOff	:= true;
end_if;

END_FUNCTION_BLOCK

(* ---- Fb_Can_Axis_Parameters.st ---- *)
(*[[
    UserText1= "V15.7",
]]*)
FUNCTION_BLOCK Fb_Can_Axis_Parameters

 	#IMPORT  "Gv_Allprocess.gvl"

VAR_INPUT
	CHN			: int;
	Node_index	: int;
	Node_Id		: int;
END_VAR

VAR_OUTPUT
    o_Status   : Dword;	(* Fb output error if 0 all is done correctly	*)
END_VAR

VAR
    la_Sline	: STRING;	(* Singol file line                             *)
    la_FieldName: STRING;   (* CAMPO DI COMANDI DA ESEGUIRE                 *)
    li_Match	: int;      (* mach string output							*)
    li_Match_1	: int;      (* mach string output <NODE_					*)
	li_ind		: int;
    ld_Tmp		: lreal;
	filehnd		: F_SYNC_FILE;
	lb_filestat	: bool;

END_VAR

(* Found in the file the key 'AXIS PARAM' *)
(* RICERCA DELLA PAROLA CHIAVE 'la_FieldName' *)
la_FieldName := CONCAT('<NODE_',INT_TO_STRING(Node_Id),
						'.',
						INT_TO_STRING(CHN),
						'>'
					   );

filehnd.FILENAME	:= CONCAT(gaIOFilePath, '\cancfg.txt');
filehnd.MODE        := CF_READ;
filehnd.POSITION    := 0;
filehnd.LSTERRCD    := 0;
filehnd.ISOPEN      := 0;

lb_filestat := F_SYNC_OPENFILE(filehnd);
if lb_filestat then
    o_Status := 1;
    RETURN;
end_if;

(* found the key <NODE_n.chn> *)
REPEAT
	lb_filestat := F_SYNC_READLINE(filehnd, la_Sline);

    if filehnd.POSITION = -1 then
        o_Status := 1;
		lb_filestat := F_SYNC_CLOSEFILE(filehnd);
        RETURN;
    end_if;

    li_Match := FIND(la_Sline, la_FieldName);
    UNTIL li_Match <> 0
end_repeat;

REPEAT
	lb_filestat := F_SYNC_READLINE(filehnd, la_Sline);
    if (filehnd.POSITION = -1) or (li_Match_1 = 0) then
        o_Status := 1;
		lb_filestat := F_SYNC_CLOSEFILE(filehnd);
        RETURN;
    end_if;
    li_Match := FIND(la_Sline, '<AXIS PARAM>');
	li_Match_1 := FIND(la_Sline, '<NODE_');
    UNTIL li_Match <> 0
end_repeat;

(* Increment the numbers of canopen motors *)
li_ind := Gi_Can_Num_Motor + 1;
GI_Can_CobidMotor[li_ind] := Node_index;
Gst_CanMotor[Node_index].CHN := CHN;
Gst_CanMotor[Node_index].NODE_ID := Node_Id;

(* Set requet to initialize the motor *)
Gst_CanMotor[Node_index].INIT := TRUE;

(* Until the key 'END' is not found analize the file *)
while (TRUE) do
    li_Match := 0;
	lb_filestat := F_SYNC_READLINE(filehnd, la_Sline);
    if filehnd.POSITION = -1 then
        o_Status := 1;
		lb_filestat := F_SYNC_CLOSEFILE(filehnd);
		Gi_Can_Num_Motor := li_ind;
        exit;
    end_if;

    li_Match := FIND(la_Sline, '<END>');
    if li_Match <> 0 then
        (* COSTANTE DI CONVERSIONE DELLA VELOCITA' DA MM/MIN A GIRI/MIN *)
        (* PER SM137 è IN GIRI/MINUTO                                   *)
        Gst_CanMotor[Node_index].VEL_CONV := 1.0/Gst_CanMotor[Node_index].ME_PITCH;

        (* Calcolo il fattore di conversione da impulsi motore a millimetri *)
        Gst_CanMotor[Node_index].POS_CONV := Gst_CanMotor[Node_index].ME_PITCH / Gst_CanMotor[Node_index].EL_PITCH;

		(* if the process is zero the cam motor is assigned at the process 1 *)
		if Gst_CanMotor[Node_index].ProcessNum = 0 then
			Gst_CanMotor[Node_index].ProcessNum := 1;
		end_if;

        o_Status := 0;
		Gi_Can_Num_Motor := li_ind;

        exit;
    end_if;

    (* Device type                        *)
    li_Match := FIND(la_Sline, '<DEVICE TYPE>') ;
    if li_Match <> 0 then
        Fn_StringToLrealB10(la_Sline, ld_Tmp);
    	Gst_CanMotor[Node_Index].DevType := lreal_to_int(ld_Tmp);
    end_if;

    (* ELECTRICAL PITCH                   *)
    li_Match := FIND(la_Sline, '<ELECTRICAL PITCH>') ;
    if li_Match <> 0 then
        Fn_StringToLrealB10(la_Sline, ld_Tmp);
    	Gst_CanMotor[Node_Index].EL_PITCH := ld_Tmp;
    end_if;

    (* MECCANICAL PITCH                  *)
    li_Match := FIND(la_Sline, '<MECCANICAL PITCH>') ;
    if li_Match <> 0 then
        Fn_StringToLrealB10(la_Sline, ld_Tmp);
    	Gst_CanMotor[Node_Index].ME_PITCH := ld_Tmp;
    end_if;

    (* TOLLERANCE SPACE   *)
    li_Match := FIND(la_Sline, '<TOLLERANCE SPACE>') ;
    if li_Match <> 0 then
        Fn_StringToLrealB10(la_Sline, ld_Tmp);
    	Gst_CanMotor[Node_Index].POSIZ_Band := ld_Tmp;
    end_if;

    (* TOLLERANCE WINDOW        *)
    li_Match := FIND(la_Sline, '<TOLLERANCE WINDOW>') ;
    if li_Match <> 0 then
        Fn_StringToLrealB10(la_Sline, ld_Tmp);
        ld_Tmp := ld_Tmp * 1000.0; (* CONVERTE IL TEMPO DA SECONDI A MILLISECONDI *)
        Gst_CanMotor[Node_Index].POSIZ_WINDOW := lreal_to_time(ld_Tmp);
    end_if;

    (* TOLLERANCE TIMEOUT              *)
    li_Match := FIND(la_Sline, '<TOLLERANCE TIMEOUT>') ;
    if li_Match <> 0 then
        Fn_StringToLrealB10(la_Sline, ld_Tmp);
        ld_Tmp := ld_Tmp * 1000.0; (* CONVERTE IL TEMPO DA SECONDI A MILLISECONDI *)
        Gst_CanMotor[Node_Index].POSIZ_TIMEOUT := lreal_to_time(ld_Tmp);
    end_if;

    (* RAPID VELOCITY                               *)
    li_Match := FIND(la_Sline, '<RAPID VELOCITY>') ;
    if li_Match <> 0 then
        Fn_StringToLrealB10(la_Sline, ld_Tmp);
        Gst_CanMotor[Node_Index].VEL_RAP := ld_Tmp;
    end_if;

    (* MANUAL VELOCITY                              *)
    li_Match := FIND(la_Sline, '<MANUAL VELOCITY>') ;
    if li_Match <> 0 then
        Fn_StringToLrealB10(la_Sline, ld_Tmp);
        Gst_CanMotor[Node_Index].VEL_MAN := ld_Tmp;
    end_if;

    (* RAPID ACCELERATION                           *)
    li_Match := FIND(la_Sline, '<RAPID ACCELERATION>') ;
    if li_Match <> 0 then
        Fn_StringToLrealB10(la_Sline, ld_Tmp);
        Gst_CanMotor[Node_Index].ACC_RAP := ld_Tmp;
    end_if;

    (* MANUAL ACCELERATION                          *)
    li_Match := FIND(la_Sline, '<MANUAL ACCELERATION>') ;
    if li_Match <> 0 then
        Fn_StringToLrealB10(la_Sline, ld_Tmp);
        Gst_CanMotor[Node_Index].ACC_MAN := ld_Tmp;
    end_if;

    (* HOMING DIRECTION  0=POSITIVO 1=NEG      *)
    li_Match := FIND(la_Sline, '<HOMING DIRECTION>') ;
    if li_Match <> 0 then
        Fn_StringToLrealB10(la_Sline, ld_Tmp);
        Gst_CanMotor[Node_Index].DIR_HOMING := (ld_Tmp = 0.0);
    end_if;

    (* POSITIVE LIMIT                        *)
    li_Match := FIND(la_Sline, '<POSITIVE LIMIT>') ;
    if li_Match <> 0 then
        Fn_StringToLrealB10(la_Sline, ld_Tmp);
        Gst_CanMotor[Node_Index].LIMOP_POS := ld_Tmp;
    end_if;

    (* NEGATIVE LIMIT                         *)
    li_Match := FIND(la_Sline, '<NEGATIVE LIMIT>') ;
    if li_Match <> 0 then
        Fn_StringToLrealB10(la_Sline, ld_Tmp);
        Gst_CanMotor[Node_Index].LIMOP_NEG := ld_Tmp;
    end_if;

    (* HOME POSITION                                   *)
    li_Match := FIND(la_Sline, '<HOME POSITION>') ;
    if li_Match <> 0 then
        Fn_StringToLrealB10(la_Sline, ld_Tmp);
        Gst_CanMotor[Node_Index].HOME_POSITION := ld_Tmp;
    end_if;

    (* HOMING VELOCITY                               *)
    li_Match := FIND(la_Sline, '<HOMING VELOCITY>') ;
    if li_Match <> 0 then
        Fn_StringToLrealB10(la_Sline, ld_Tmp);
        Gst_CanMotor[Node_Index].VEL_HOMING := ld_Tmp;
    end_if;

    (* Address of info to handle the motor *)
	(* Can PDO Control word offset in bytes *)
    li_Match := FIND(la_Sline, '<RPDO_CW_OFFSET>') ;
    if li_Match <> 0 then
        Fn_StringToLrealB10(la_Sline, ld_Tmp);
        Gst_CanMotor[Node_Index].INDCW := lreal_to_int(ld_Tmp);
    end_if;

    li_Match := FIND(la_Sline, '<RPDO_POSITION_OFFSET>') ;
    if li_Match <> 0 then
        Fn_StringToLrealB10(la_Sline, ld_Tmp);
        Gst_CanMotor[Node_Index].INDPOS := lreal_to_int(ld_Tmp);
    end_if;

    li_Match := FIND(la_Sline, '<RPDO_OPMODE_OFFSET>') ;
    if li_Match <> 0 then
        Fn_StringToLrealB10(la_Sline, ld_Tmp);
        Gst_CanMotor[Node_Index].INDMODOCN := lreal_to_int(ld_Tmp);
    end_if;

    li_Match := FIND(la_Sline, '<RPDO_VELOCITY_OFFSET>') ;
    if li_Match <> 0 then
        Fn_StringToLrealB10(la_Sline, ld_Tmp);
        Gst_CanMotor[Node_Index].IND_VEL := lreal_to_int(ld_Tmp);
    end_if;

    li_Match := FIND(la_Sline, '<TPDO_SW_OFFSET>') ;
    if li_Match <> 0 then
        Fn_StringToLrealB10(la_Sline, ld_Tmp);
        Gst_CanMotor[Node_Index].INDSW := lreal_to_int(ld_Tmp);
    end_if;

    li_Match := FIND(la_Sline, '<TPDO_MOTOR_ENCODER_OFFSET>') ;
    if li_Match <> 0 then
        Fn_StringToLrealB10(la_Sline, ld_Tmp);
        Gst_CanMotor[Node_Index].INDPOS_INP := lreal_to_int(ld_Tmp);
    end_if;

    li_Match := FIND(la_Sline, '<TPDO_ACT_OPMODE_OFFSET>') ;
    if li_Match <> 0 then
        Fn_StringToLrealB10(la_Sline, ld_Tmp);
        Gst_CanMotor[Node_Index].INDMODOMOT := lreal_to_int(ld_Tmp);
    end_if;

    li_Match := FIND(la_Sline, '<TPDO_ACT_TORQUE_OFFSET>') ;
    if li_Match <> 0 then
        Fn_StringToLrealB10(la_Sline, ld_Tmp);
        Gst_CanMotor[Node_Index].INDTORQUE := lreal_to_int(ld_Tmp);
    end_if;

	(* INDEX OF THE PREVIOUS MOTOR TO CHECK OPERATIVE LIMIT and COLLISION *)
    li_Match := FIND(la_Sline, '<PREVIOUS MOTOR NUMBER>') ;
    if li_Match <> 0 then
        Fn_StringToLrealB10(la_Sline, ld_Tmp);
        Gst_CanMotor[Node_Index].PREV_MOTOR_INDEX := lreal_to_int(ld_Tmp);
    end_if;

	(* INDEX OF THE PREVIOUS MOTOR TO CHECK OPERATIVE LIMIT and COLLISION *)
    li_Match := FIND(la_Sline, '<NEXT MOTOR NUMBER>') ;
    if li_Match <> 0 then
        Fn_StringToLrealB10(la_Sline, ld_Tmp);
        Gst_CanMotor[Node_Index].NEXT_MOTOR_INDEX := lreal_to_int(ld_Tmp);
    end_if;

	(* BREAKE ACTIVE *)
    li_Match := FIND(la_Sline, '<MOTOR WITH BREAKE>') ;
    if li_Match <> 0 then
        Fn_StringToLrealB10(la_Sline, ld_Tmp);
        Gst_CanMotor[Node_Index].BREAKE := (ld_Tmp <> 0.0);;
    end_if;

	(* NULL OFFSET *)
    li_Match := FIND(la_Sline, '<NULL OFFSET>') ;
    if li_Match <> 0 then
        Fn_StringToLrealB10(la_Sline, ld_Tmp);
        Gst_CanMotor[Node_Index].NULL_OFFSET := ld_Tmp;
    end_if;

	(* BACK LASH *)
    li_Match := FIND(la_Sline, '<BACK LASH>') ;
    if li_Match <> 0 then
        Fn_StringToLrealB10(la_Sline, ld_Tmp);
        Gst_CanMotor[Node_Index].BACK_LASH := ld_Tmp;
    end_if;

	(* Motor is on table number ... *)
    li_Match := FIND(la_Sline, '<MOTOR ON TABLE>') ;
    if li_Match <> 0 then
        Fn_StringToLrealB10(la_Sline, ld_Tmp);
        Gst_CanMotor[Node_Index].TABLE := lreal_to_int(ld_Tmp);
    end_if;

end_while;

lb_filestat := F_SYNC_CLOSEFILE(filehnd);

END_FUNCTION_BLOCK
